// TIA Portal V19 export
ORGANIZATION_BLOCK "Main"   // OB1, LAD, ProgramCycle
{ S7_Optimized_Access := 'TRUE' }
// stored: SetENOAutomatically false
   VAR_INPUT
      Initial_Call : Bool;
      Remanence : Bool;
   END_VAR
BEGIN

REGION Network 1
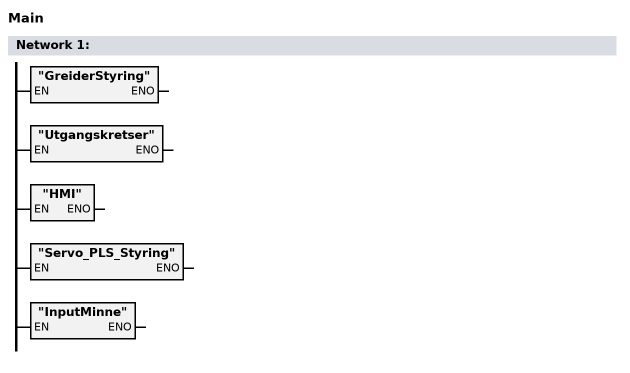
   RUNG wire#powerrail
      "GreiderStyring"()
   END_RUNG
   RUNG wire#powerrail
      "Utgangskretser"()
   END_RUNG
   RUNG wire#powerrail
      "HMI"()
   END_RUNG
   RUNG wire#powerrail
      "Servo_PLS_Styring"()
   END_RUNG
   RUNG wire#powerrail
      "InputMinne"()
   END_RUNG
   // the same network as SCL:
   "GreiderStyring"();
   "Utgangskretser"();
   "HMI"();
   "Servo_PLS_Styring"();
   "InputMinne"();
END_REGION
END_ORGANIZATION_BLOCK
